FUNCTION_BLOCK INTERNAL FB_ArrayHelper_Tests EXTENDS FB_TestSuite
VAR_INPUT
END_VAR
VAR_OUTPUT
END_VAR

Test01_GetArrayElementCount();
Test02_GetArrayMaxIndex();
Test03_InsertNumber();
Test04_InsertString();
Test05_InsertStruct();
Test06_ShiftUp_ExpectLastElementOverwriteFirstElementZero();
Test07_SetAtFirstEmptySlot();
Test08_AllMethods_provideNonArrayVar_ExpectNothing();
Test09_InsertIntoEmptyArray_ExpectOnlyFirstItem();
Test10_CheckIfArrayContainsItem();
Test11_ClearArray_ExpectEmptyArray();
Test12_ReferenceToArrayWithAllMethods_ExpectNormalResults();
Test13_FindLastOccupiedItem();
Test14_ShiftDown_ExpectFirstElementOverwriteLastElementZero();

METHOD Test01_GetArrayElementCount
VAR_INPUT
END_VAR
VAR
	arr		: ARRAY[0..99] OF REAL;
	arr2	: ARRAY[22..33] OF REAL;
END_VAR
TcUnit.TEST('Test01_GetArrayElementCount');

AssertEquals_DINT(
	Actual := ArrayHelper.GetElementCount(arr := arr, dataType := arr[0]),
	Expected := 100,
	Message := 'Getting array element count failed!');
	
AssertEquals_DINT(
	Actual := ArrayHelper.GetElementCount(arr := arr2, dataType := arr2[22]),
	Expected := 33 - 22 + 1,
	Message := 'Getting array element count for array with non-zero start element index failed!');
	
TcUnit.TEST_FINISHED();
END_METHOD

METHOD Test02_GetArrayMaxIndex
VAR_INPUT
END_VAR
VAR
	arr		: ARRAY[0..99] OF REAL;
	arr2	: ARRAY[22..33] OF REAL;
END_VAR
TcUnit.TEST('Test02_GetArrayMaxIndex');

AssertEquals_DINT(
	Actual := ArrayHelper.GetMaxIndex(arr := arr, dataType := arr[0], startIndex := 0),
	Expected := 99,
	Message := 'Getting array maximum index failed!');
	
AssertEquals_DINT(
	Actual := ArrayHelper.GetMaxIndex(arr := arr2, dataType := arr2[22], startIndex := 22),
	Expected := 33,
	Message := 'Getting array maximum index for array with non-zero start element index failed!');
	
TcUnit.TEST_FINISHED();
END_METHOD

METHOD PRIVATE Test03_InsertNumber
VAR_INPUT
END_VAR

VAR
	i		: INT;
	value	: INT := 99;
	arr		: ARRAY [0..10] OF INT;
END_VAR
TcUnit.TEST('Test03_InsertNumber');

FOR i := 0 TO 10 BY 1 DO
	arr[i] := i;
END_FOR

ArrayHelper.InsertAtStart(
	arr := arr,
	item := value);
	
AssertEquals_INT(
	Expected := value,
	Actual := arr[0],
	Message := 'First item was not inserted properly!');
	
AssertEquals_INT(
	Expected := 9,
	Actual := arr[10],
	Message := 'Last item was not removed from the array!!');
	
TcUnit.TEST_FINISHED();
END_METHOD

METHOD PRIVATE Test04_InsertString
VAR_INPUT
END_VAR

VAR
	i		: INT;
	value	: STRING := '9';
	arr		: ARRAY [0..10] OF STRING;
END_VAR
TcUnit.TEST('Test04_InsertString');

FOR i := 0 TO 10 BY 1 DO
	arr[i] := INT_TO_STRING(i);
END_FOR

ArrayHelper.InsertAtStart(
	arr := arr,
	item := value);
	
AssertEquals_STRING(
 	Actual:= arr[0],
	Expected := value,
	Message := 'First item was not inserted properly!');
	
AssertEquals_STRING(
	Expected := '9',
	Actual := arr[10],
	Message := 'Last item was not removed from the array!!');
	
TcUnit.TEST_FINISHED();
END_METHOD

METHOD Test05_InsertStruct

VAR
	i		: INT;
	value	: ST_GenericError;
	arr		: ARRAY [0..10] OF ST_GenericError;
END_VAR
TcUnit.TEST('Test05_InsertStruct');

FOR i := 0 TO 10 BY 1 DO
	arr[i].Code := i;
	arr[i].Message := INT_TO_STRING(i);
END_FOR

ArrayHelper.InsertAtStart(
	arr := arr,
	item := value);
	
AssertEquals(
	Expected := value,
	Actual := arr[0],
	Message := 'First item was not inserted properly!');
	
AssertEquals_STRING(
	Expected := '9',
	Actual := arr[10].Message,
	Message := 'Last item was not removed from the array!');
	
AssertEquals_STRING(
	Expected := '9',
	Actual := arr[10].Message,
	Message := 'Last item was not removed from the array!');
	
TcUnit.TEST_FINISHED();
END_METHOD

METHOD Test06_ShiftUp_ExpectLastElementOverwriteFirstElementZero
VAR_INPUT
END_VAR

VAR_INST
	arr	: ARRAY[0..20] OF INT;
	i	: int;
END_VAR
TcUnit.TEST('Test06_ShiftUp_ExpectLastElementOverwriteFirstElementZero');

FOR i := 0 TO 20 BY 1 DO
	arr[i] := i;
END_FOR

ArrayHelper.ShiftUp(
	arr := arr,
	dataType := arr[0]);
AssertEquals_INT(
	Actual := arr[0],
	Expected := 0,
	Message := 'Shifting the array up, first element should be set to 0!');
	
FOR i := 1 TO 20 BY 1 DO
	AssertEquals_INT(
		Actual := arr[i],
		Expected := i-1,
		Message := Tc2_Standard.CONCAT('Shifting up failed! Incorrect value at position ', TO_STRING(i)));
END_FOR
	
TcUnit.TEST_FINISHED();
END_METHOD

METHOD Test07_SetAtFirstEmptySlot
VAR_INPUT
END_VAR

VAR
	arr		: ARRAY[0..69] OF T_ArrayIndexer;
	arr2	: ARRAY[0..69] OF BOOL;
	valueToSet	: T_ArrayIndexer := 9999;
	i	: T_ArrayIndexer;
	boolValueToSet	: BOOL := TRUE;
END_VAR
TcUnit.TEST('Test07_SetAtFirstEmptySlot');

FOR i := 0 TO 30 BY 1 DO
	arr[i] := i + 1;
	arr2[i] := TRUE;
END_FOR

ArrayHelper.SetAtFirstEmptySlot(
	arr := arr,
	item := valueToSet);

ArrayHelper.SetAtFirstEmptySlot(
	arr := arr2,
	item := boolValueToSet);

FOR i := 0 TO 30 BY 1 DO
	AssertEquals_DINT(
		Expected := i + 1,
		Actual := arr[i],
		Message := 'Setting first empty slot should not have changed non-empty fields!');
		
	AssertTrue(
		Condition := arr2[i],
		Message := 'Setting first empty slot for array of booleans should not have changed non-empty fields!');
END_FOR

AssertEquals(
	Expected := valueToSet,
	Actual := arr[31],
	Message := 'Setting first empty slot failed, first empty element differs!');
	
AssertTrue(
	Condition := arr2[31],
	Message := 'Setting first empty slot failed, first empty element should be set to TRUE!');
	
AssertEquals_DINT(
	Expected := 0,
	Actual := arr[32],
	Message := 'Setting first empty slot failed, item after the inserted slot should be empty!');
	
AssertFalse(
	Condition := arr2[32],
	Message := 'Setting first empty slot failed, item after the inserted slot should be empty!');	
	

TcUnit.TEST_FINISHED();
END_METHOD

METHOD Test08_AllMethods_provideNonArrayVar_ExpectNothing
VAR_INPUT
END_VAR
VAR
	notAnArray	: BOOL := TRUE;
	val			: BOOL;
END_VAR
TcUnit.TEST('Tes08_AllMethods_provideNonArrayVar_ExpectNothing');

ArrayHelper.GetElementCount(arr := notAnArray, dataType := val);
AssertTrue(
	Condition := notAnArray, 
	Message := 'When non-array is provided to any method, the method should not execute anything!');

AssertEquals_DINT(
	Actual := ArrayHelper.GetMaxIndex(arr := notAnArray, dataType := val, startIndex := 0),
	Expected := 0,
	Message := 'When non-array is provided, max index returned should be 0!');
	
AssertTrue(
	Condition := notAnArray, 
	Message := 'When non-array is provided to any method, the method should not execute anything!');

	
TcUnit.TEST_FINISHED();
END_METHOD

METHOD Test09_InsertIntoEmptyArray_ExpectOnlyFirstItem
VAR_INPUT
END_VAR

VAR_INST
	arr			: ARRAY[0..20] OF ST_GenericError;
	item		: ST_GenericError := (Code := 0, Message := '0');
	emptyItem	: ST_GenericError;
	i 			: T_ArrayIndexer;
END_VAR
TcUnit.TEST('Test09_InsertIntoEmptyArray_ExpectOnlyFirstItem');

FOR i := 0 TO 20 BY 1 DO
	AssertEquals(Actual := arr[i], Expected := emptyItem, Message := 'Wrong array initialization!');
END_FOR

ArrayHelper.InsertAtStart(arr := arr, item := item);

AssertEquals(
	Actual := arr[0], 
	Expected := item, 
	Message := 'InsertAtStart should have first item in array the same as item being inserted!');
	
FOR i := 1 TO 20 BY 1 DO
	AssertEquals(Actual := arr[i], Expected := emptyItem, 
		Message := Tc2_Standard.CONCAT(
			STR1 := 'InsertAtStart should have left other elements unchanged! Changed element at index ', 
			STR2 := TO_STRING(i) ));
END_FOR

ArrayHelper.InsertAtStart(arr := arr, item := item);
AssertEquals(
	Actual := arr[0], 
	Expected := item, 
	Message := 'Inserting at start for the second time - 1st item is incorrect!');
AssertEquals(
	Actual := arr[1], 
	Expected := item, 
	Message := 'Inserting at start for the second time - 2nd item is incorrect!');	

TcUnit.TEST_FINISHED();
END_METHOD

METHOD Test10_CheckIfArrayContainsItem
VAR_INST
	arr		: ARRAY[0..10] OF STRING;
	item	: STRING := 'mwah';
END_VAR
TcUnit.TEST('Test10_CheckIfArrayContainsItem');

ArrayHelper.Clear(arr);
AssertFalse(
	Condition := ArrayHelper.DoesArrayContainItem(arr, item),
	Message := 'Array does not contain the item, method should return FALSE.');

arr[0] := item;

AssertTrue(
	Condition := ArrayHelper.DoesArrayContainItem(arr, item),
	Message := 'Array does contain the item on 0th index, method should return TRUE.');
	
arr[0] := '';
arr[5] := item;

AssertTrue(
	Condition := ArrayHelper.DoesArrayContainItem(arr, item),
	Message := 'Array does contain the item on 5th index, method should return TRUE.');
	
arr[5] := '';
arr[10] := item;	
AssertTrue(
	Condition := ArrayHelper.DoesArrayContainItem(arr, item),
	Message := 'Array does contain the item on 10th index, method should return TRUE.');

arr[0] := 'lalala';
arr[3] := 'aahah';
AssertTrue(
	Condition := ArrayHelper.DoesArrayContainItem(arr, item),
	Message := 'Array does contain the item on 10th index, but also includes non empty elements before, method should return TRUE.');

arr[2] := item;
AssertTrue(
	Condition := ArrayHelper.DoesArrayContainItem(arr, item),
	Message := 'Array does contain the item on 2nd index, but also includes non empty elements before and after, method should return TRUE.');	
	
TcUnit.TEST_FINISHED();
END_METHOD

METHOD Test11_ClearArray_ExpectEmptyArray
VAR_INPUT
END_VAR
VAR_INST
	arrUnmodified	: ARRAY[0..20] OF BOOL;
	arrModified		: ARRAY[0..20] OF BOOL;
	idx				: T_ArrayIndexer;
END_VAR
TcUnit.TEST('Test11_ClearArray_ExpectEmptyArray');

FOR idx := 0 TO 20 BY 1 DO
	arrModified[idx] := TRUE;
END_FOR

AssertTrue(
	Condition := ArrayHelper.Clear(arrModified),
	Message := 'Clearing array returned FALSE when it should have been TRUE.');

AssertArrayEquals_BOOL(
	Actuals := arrModified,
	Expecteds := arrUnmodified,
	Message := 'Array contents were not cleared.');

TcUnit.TEST_FINISHED();
END_METHOD

METHOD Test12_ReferenceToArrayWithAllMethods_ExpectNormalResults
VAR_INST
	arr			: ARRAY[0..10] OF REAL;
	refArr		: REFERENCE TO ARRAY[0..10] OF REAL;
	arrEmpty	: ARRAY[0..10] OF REAL;
	findResult	: REAL;
END_VAR
TcUnit.TEST('Test12_ReferenceToArrayWithAllMethods_ExpectNormalResults');
refarr REF= arr;
arr[5] := 22.2;

ArrayHelper.Clear(refArr);
AssertArrayEquals_REAL(
	Actuals := arr,
	Expecteds := arrEmpty,
	Delta := 0,
	Message := 'Clear array failed.');
	
arr[6] := 5.3;
AssertTrue(
	Condition := ArrayHelper.DoesArrayContainItem(arr := refArr, item := arr[6]),
	Message := 'DoesArrayContainItem failed.');

AssertTrue(
	Condition := ArrayHelper.FindLastOccupiedItem(refArr, refArr[0], findResult),
	Message := 'FindLastOccupiedItem failed (returned FALSE).');

AssertEquals_REAL(
	Actual := findResult,
	Expected := 5.3,
	Delta := 0,
	Message := 'FindLastOccupiedItem output value was incorrect.');
	
AssertEquals_DINT(
	Actual := ArrayHelper.GetElementCount(refArr, refArr[0]),
	Expected := 11,
	Message := 'GetEleeentCount failed.');
	
AssertEquals_DINT(
	Actual := ArrayHelper.GetMaxIndex(refArr, refArr[0], 0),
	Expected := 10,
	Message := 'GetMaxIndex failed.');
	
ArrayHelper.InsertAtStart(refArr, findResult);
AssertEquals_REAL(
	Actual := refArr[0],
	Expected := 5.3,
	Delta := 0.0,
	Message := 'InsertAtStart failed');

arr[0] := 0;	
ArrayHelper.SetAtFirstEmptySlot(refArr, findResult);	
AssertEquals(
	Expected := findResult,
	Actual := refArr[0],
	Message := 'SetAtFirstEmptySlot failed.');
	
arr[1] := 5.5;
ArrayHelper.ShiftDown(refArr, refArr[0]);
AssertEquals_REAL(
	Actual := refArr[0],
	Expected := 5.5,
	Delta := 0.0,
	Message := 'ShiftDown failed.');

ArrayHelper.ShiftUp(refARr, refArr[0]);
AssertEquals_REAL(
	Actual := refArr[1],
	Expected := 5.5,
	Delta := 0.0,
	Message := 'ShiftUp failed.');

TcUnit.TEST_FINISHED();
END_METHOD

METHOD Test13_FindLastOccupiedItem
VAR_INPUT
END_VAR

VAR_INST
	arr	: ARRAY[0..10] OF INT;
	result	: int;
END_VAR
TcUnit.TEST('Test13_FindLastOccupiedItem');

AssertFalse(
	Condition := ArrayHelper.FindLastOccupiedItem(arr, arr[0], result),
	Message := 'Empty array should return FALSE.');
	
arr[5] := 5;

AssertTrue(	
	Condition := ArrayHelper.FindLastOccupiedItem(arr, arr[0], result),
	Message := 'Expected TRUE, 5th element is not empty.');
	
AssertEquals_INT(
	Actual := result,
	Expected := 5,
	Message := 'Incorrect result when finding last occupied element.');
	
TcUnit.TEST_FINISHED();
END_METHOD

METHOD Test14_ShiftDown_ExpectFirstElementOverwriteLastElementZero
VAR_INPUT
END_VAR

VAR
	arr	: ARRAY[0..20] OF INT;
	i	: int;
END_VAR
TcUnit.TEST('Test14_ShiftDown_ExpectFirstElementOverwriteLastElementZero');

FOR i := 0 TO 20 BY 1 DO
	arr[i] := i;
END_FOR

ArrayHelper.ShiftDown(
	arr := arr,
	dataType := arr[0]);
	
AssertEquals_INT(
	Actual := arr[20],
	Expected := 0,
	Message := 'Shifting the array down, last element should be set to 0!');
	
FOR i := 19 TO 0 BY -1 DO
	AssertEquals_INT(
		Actual := arr[i],
		Expected := i+1,
		Message := Tc2_Standard.CONCAT('Shifting up failed! Incorrect value at position ', TO_STRING(i)));
END_FOR
	
TcUnit.TEST_FINISHED();
END_METHOD

END_FUNCTION_BLOCK

(* stored: Version 1.1.0.1, ProductVersion 3.1.4024.15
   POU FB_ArrayHelper_Tests: Id {6e9b477f-91da-07b8-384b-0f33de518108}, SpecialFunc None
   Method Test01_GetArrayElementCount: Id {2f0a8400-5b23-0ca4-3735-368e9840cbd2}
   Method Test02_GetArrayMaxIndex: Id {bc1d8f1a-639c-0a77-144a-0a527e117e1d}
   Method Test03_InsertNumber: Id {0bc2a11d-75c0-04a1-3c2e-0d3eb1417ca6}
   Method Test04_InsertString: Id {df991e0c-a369-0719-2350-4b8343f2f03b}
   Method Test05_InsertStruct: Id {f4b22831-ae98-024d-016e-1c50385778ff}
   Method Test06_ShiftUp_ExpectLastElementOverwriteFirstElementZero: Id {67ea1074-796a-03e4-1529-5e485181dbca}
   Method Test07_SetAtFirstEmptySlot: Id {378655a2-db0d-0d65-1026-2faa831ee346}
   Method Test08_AllMethods_provideNonArrayVar_ExpectNothing: Id {3ee8021c-32e6-0293-3123-601800a244ac}
   Method Test09_InsertIntoEmptyArray_ExpectOnlyFirstItem: Id {a8d8434e-596a-00a0-21e3-47c7bf1b2911}
   Method Test10_CheckIfArrayContainsItem: Id {35878296-f39d-0da2-34a7-e3adc7bd6e85}
   Method Test11_ClearArray_ExpectEmptyArray: Id {cc53d4a8-f18c-0f01-352b-998b267791ec}
   Method Test12_ReferenceToArrayWithAllMethods_ExpectNormalResults: Id {347793f1-d4c3-04a6-364e-b7ee092ed247}
   Method Test13_FindLastOccupiedItem: Id {2fe3197e-d9e2-07ac-3526-3dff66a0a860}
   Method Test14_ShiftDown_ExpectFirstElementOverwriteLastElementZero: Id {e80b21d9-d3f9-0ea9-07b5-130b5201d4b3} *)
